PROGRAM MAIN
VAR

	trigger: BOOL;
	
END_VAR

IF trigger THEN
	
	trigger := FALSE;
	
	ADSLOGSTR( 
		msgCtrlMask := ADSLOG_MSGTYPE_ERROR OR ADSLOG_MSGTYPE_MSGBOX,
        msgFmtStr := 'This is a test message : %s', 
		strArg := '123'
	);
		
END_IF

END_PROGRAM

(* stored: Version 1.1.0.1, ProductVersion 3.1.4024.9
   POU MAIN: Id {51ec683b-10ce-43eb-9703-c0633aae0bfd}, SpecialFunc None *)
